(* IEC 61131-3 sources: plc_generation_empirical_study/datasets/_archive/pre_native_plcverif_20260810/tasks/C03_H02_safety_zone_arbitration, 2 files *)

(* ---- interface.st ---- *)
FUNCTION_BLOCK C03_H02_safety_zone_arbitration
VAR_INPUT
    RobotRequest : BOOL;
    ConveyorRequest : BOOL;
    ManualRequest : BOOL;
    GuardClosed : BOOL;
    EStopOK : BOOL;
    ManualKey : BOOL;
END_VAR
VAR_OUTPUT
    RobotEnable : BOOL;
    ConveyorEnable : BOOL;
    ManualEnable : BOOL;
    Conflict : BOOL;
END_VAR
END_FUNCTION_BLOCK

(* ---- reference.st ---- *)
FUNCTION_BLOCK C03_H02_safety_zone_arbitration
VAR_INPUT
    RobotRequest : BOOL;
    ConveyorRequest : BOOL;
    ManualRequest : BOOL;
    GuardClosed : BOOL;
    EStopOK : BOOL;
    ManualKey : BOOL;
END_VAR
VAR_OUTPUT
    RobotEnable : BOOL;
    ConveyorEnable : BOOL;
    ManualEnable : BOOL;
    Conflict : BOOL;
END_VAR

RobotEnable := FALSE;
ConveyorEnable := FALSE;
ManualEnable := FALSE;
Conflict := (RobotRequest AND ConveyorRequest)
            OR (RobotRequest AND ManualRequest AND ManualKey)
            OR (ConveyorRequest AND ManualRequest AND ManualKey);

IF GuardClosed AND EStopOK THEN
    IF ManualRequest AND ManualKey THEN
        ManualEnable := TRUE;
    ELSIF RobotRequest THEN
        RobotEnable := TRUE;
    ELSIF ConveyorRequest THEN
        ConveyorEnable := TRUE;
    END_IF;
END_IF;

END_FUNCTION_BLOCK
